(* CoDeSys 2.3.8.0 project: RetMemory_BX.prx *)
(* Libraries: STANDARD.LBX 5.12.03 08:02:30 *)

(* Task configuration *)
TASK Standard (PRIORITY := 0, INTERVAL := T#20ms);
	MAIN
END_TASK

(* POU MAIN, CFC *)
PROGRAM MAIN
VAR
	fbStore: FB_StoreMemory;
	Array_Memory AT %MB0: ARRAY [0..20] OF WORD;
END_VAR
VAR RETAIN PERSISTENT
	Array_Retain: ARRAY [0..20] OF WORD; (*Zmienne przechowywane w sterowniku  -sposób deklaracji, przechowywania zależny od sterownika*)
END_VAR
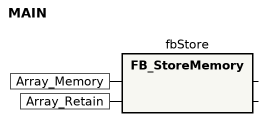
_CFC_ (* Continuous Function Chart, elements in execution order *)
#0 fbStore:FB_StoreMemory(Array_Memory, Array_Retain)
_END_CFC_
(* the same logic as Structured Text *)
fbStore(Array_Memory, Array_Retain);
END_PROGRAM

(* POU FB_StoreMemory, ST *)
FUNCTION_BLOCK FB_StoreMemory
VAR_IN_OUT
	Array_Memory: ARRAY [0..20] OF WORD;
	Array_Retain: ARRAY [0..20] OF WORD;
END_VAR
VAR
	bFirstCycle: BOOL:= TRUE;
	i: BYTE;
END_VAR
IF bFirstCycle THEN(*Rozpoznanie pierwszego cyklu programu*)
	FOR i:=0 TO 20 DO
		Array_Memory[i] := Array_Retain[i];(*Przepisanie pamięci nieulotnej do tablicy memory*)
	END_FOR
ELSE
	FOR i:=0 TO 20 DO
		Array_Retain[i] := Array_Memory[i]; (*Przepisanie tablicy memory do pamięci nieulotnej*)
	END_FOR
END_IF
bFirstCycle := FALSE;
END_FUNCTION_BLOCK
